Universal Robots PolyScope program: WSG-template.urp

ProgramRoot directory=/programs/Weiss_Robotics; kinematics=(a=[0, -0.24365, -0.21325, 0, 0, 0], d=[0.1519, 0, 0, 0.11235, 0.08535, 0.0819], alpha=[1.5708, 0, 0, 1.5708, -1.5708, 0], deltaTheta=[0, 0, 0, 0, 0, 0], status=notInitialized); lastSavedInVersion=(project__name=Polyscope, major__version=3, minor__version=1, svn__revision=17336, build__date=Mar 26 2015, 11:23:02); name=WSG-template; programVersion=(project__name=Polyscope, major__version=3, minor__version=1, svn__revision=17336, build__date=Mar 26 2015, 11:23:02); robotEnvironmentFileName=WSG; serialNumberRobot=2014339999
  BeforeStart description=COMMAND_SEQUENCE_BEFORE_PROGRAM_START; name=BeforeStart
    Assignment expr=0; operatorValueType=INTEGER; valueSource=EXPRESSION
    Assignment expr=5000; operatorValueType=INTEGER; valueSource=EXPRESSION
    Assignment expr=2000; operatorValueType=INTEGER; valueSource=EXPRESSION
    Assignment expr="Idle"; operatorValueType=INTEGER; valueSource=EXPRESSION
    CallSubProgram 
    CallSubProgram 
    CallSubProgram 
    CallSubProgram 
  MainProgram cartesianAcceleration=1.2; cartesianSpeed=0.25; jointAcceleration=1.3962634015954636; jointSpeed=1.0471975511965976; sharedProcessMoveBlendRadius=0.025; motionType=JOINT_SPACE
    Placeholder 
  SubProgram [hidden by the author, left out]
  SubProgram [hidden by the author, left out]
  SubProgram [hidden by the author, left out]
  SubProgram [hidden by the author, left out]
  SubProgram [hidden by the author, left out]
  SubProgram [hidden by the author, left out]
  SubProgram [hidden by the author, left out]
  SubProgram [hidden by the author, left out]
  SubProgram [hidden by the author, left out]
  SubProgram [hidden by the author, left out]
  SubProgram [hidden by the author, left out]
